FUNCTION F_TOD_RTN : TOD
VAR_INPUT
	stArg : ST_Arg;
END_VAR
VAR
	sysVar_Info : __SYSTEM.VAR_INFO;
END_VAR

sysVar_Info := __VARINFO(F_TOD_RTN);
IF stArg.TypeClass = sysVar_Info.TypeClass THEN 
	F_TOD_RTN := TO_TOD(stArg.sValue);
	END_IF

END_FUNCTION

(* stored: Version 1.1.0.1, ProductVersion 3.1.4024.4
   POU F_TOD_RTN: Id {33804d3e-913e-4063-bc3e-c9a003f6c6fe}, SpecialFunc None *)
